// TIA Portal project "ikiyonlucal_asenkmotora_yildizucgenyolverme" (V18)

(* hardware
DEVICE "S7-1200 station_1"  S7-1200 Station
   slot 0: "Rack_0"  S7-1200 Rack  Rack  V1.0
   slot 1: "PLC_1"  CPU 1214C AC/DC/Rly  6ES7 214-1BG40-0XB0  V4.6
*)

// ===== PLC "PLC_1"  CPU 1214C AC/DC/Rly =====

VAR_GLOBAL   // PLC tag table "Default tag table"
   "STOP" AT %I0.0 : Bool;
   "İLERİ BUTON" AT %I0.1 : Bool;
   "GERİ BUTON" AT %I0.2 : Bool;
   "İLERİ KONTAKTÖR" AT %Q0.0 : Bool;
   "GERİ KONTAKTÖR" AT %Q0.1 : Bool;
   "YILDIZ KONTAKTÖR" AT %Q0.2 : Bool;
   "ÜÇGEN KONTAKTÖR" AT %Q0.3 : Bool;
END_VAR

// folder: System blocks/Program resources

DATA_BLOCK "T1"   // DB1
{ S7_Optimized_Access := 'TRUE' }
AUTHOR : Simatic
FAMILY : IEC
NAME : IEC_TMR
VERSION : 1.0
// stored: InstanceOfName IEC_TIMER
"IEC_TIMER"
BEGIN
END_DATA_BLOCK

// folder: (top level)

ORGANIZATION_BLOCK "Main"   // OB1, LAD, ProgramCycle
TITLE = "Main Program Sweep (Cycle)"
{ S7_Optimized_Access := 'TRUE' }
VERSION : 0.1
   VAR_INPUT
      Initial_Call : Bool;   // Initial call of this OB
      Remanence : Bool;   // =True, if remanent data are available
   END_VAR
BEGIN

REGION Network 1
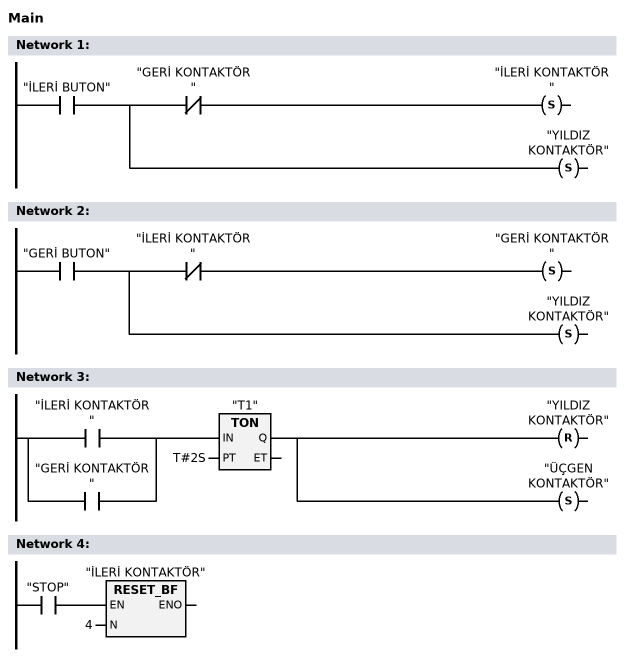
   RUNG wire#powerrail
      Contact( "İLERİ BUTON" )
      wire#w1
      I_Contact( "GERİ KONTAKTÖR" )
      S_Coil( "İLERİ KONTAKTÖR" )
   END_RUNG
   RUNG wire#w1
      S_Coil( "YILDIZ KONTAKTÖR" )
   END_RUNG
   // the same network as SCL:
   IF "İLERİ BUTON" AND NOT "GERİ KONTAKTÖR" THEN "İLERİ KONTAKTÖR" := TRUE; END_IF;
   IF "İLERİ BUTON" THEN "YILDIZ KONTAKTÖR" := TRUE; END_IF;
END_REGION

REGION Network 2
   RUNG wire#powerrail
      Contact( "GERİ BUTON" )
      wire#w1
      I_Contact( "İLERİ KONTAKTÖR" )
      S_Coil( "GERİ KONTAKTÖR" )
   END_RUNG
   RUNG wire#w1
      S_Coil( "YILDIZ KONTAKTÖR" )
   END_RUNG
   // the same network as SCL:
   IF "GERİ BUTON" AND NOT "İLERİ KONTAKTÖR" THEN "GERİ KONTAKTÖR" := TRUE; END_IF;
   IF "GERİ BUTON" THEN "YILDIZ KONTAKTÖR" := TRUE; END_IF;
END_REGION

REGION Network 3
   "T1".TON(IN := "İLERİ KONTAKTÖR" OR "GERİ KONTAKTÖR", PT := T#2S);
   IF "T1".Q THEN
       "YILDIZ KONTAKTÖR" := FALSE;
       "ÜÇGEN KONTAKTÖR" := TRUE;
   END_IF;
END_REGION

REGION Network 4
   // no SCL statement known for RBitfield: written as a call
   IF "STOP" THEN RESET_BF(operand := "İLERİ KONTAKTÖR", n := 4); END_IF;
END_REGION
END_ORGANIZATION_BLOCK